KUKA KRL program: paintImage.src, paintImage.dat

--- paintImage.src ---
&ACCESS RVP
&REL 47
DEF paintImage( )
;FOLD Declaration
   DECL EKI_STATUS RET
   DECL FRAME nextPoint
   DECL INT status
   DECL INT currentColor
   DECL BOOL pathStart
   $FLAG[1]=FALSE



   ;FOLD INI;%{PE}
      ;FOLD BASISTECH INI
         GLOBAL INTERRUPT DECL 3 WHEN $STOPMESS==TRUE DO IR_STOPM ( )
         INTERRUPT ON 3
         BAS (#INITMOV,0 )
      ;ENDFOLD (BASISTECH INI)
      ;FOLD USER INI
         ;Make your modifications here

      ;ENDFOLD (USER INI)
      ;ENDFOLD (INI)
      ;FOLD Initialize sample data
         nextPoint = {X 200,Y 600,Z 600}
         status = 0
         currentColor = 1000
         pathStart = TRUE

      ;ENDFOLD (Initialize sample data)
      ;ENDFOLD (Declaration)


   ;FOLD PTP HOME  Vel= 100 % DEFAULT;%{PE}%MKUKATPBASIS,%CMOVE,%VPTP,%P 1:PTP, 2:HOME, 3:, 5:100, 7:DEFAULT
      $BWDSTART = FALSE
      PDAT_ACT=PDEFAULT
      FDAT_ACT=FHOME
      BAS (#PTP_PARAMS,10 )
      $H_POS=XHOME
      PTP  XHOME
   ;ENDFOLD


;FOLD PTP P8 Vel=10 % PDAT4 Tool[2]:pinselC Base[3]:canvas1;%{PE}%R 8.3.48,%MKUKATPBASIS,%CMOVE,%VPTP,%P 1:PTP, 2:P8, 3:, 5:10, 7:PDAT4
$BWDSTART=FALSE
PDAT_ACT=PPDAT4
FDAT_ACT=FP8
BAS(#PTP_PARAMS,10)
PTP XP8
;ENDFOLD
RET=EKI_Init("xmlPaintImage")
RET=EKI_Open("xmlPaintImage")

LOOP
WAIT FOR $FLAG[993] == TRUE
RET=EKI_GetInt("xmlPaintImage","Ext/Status",status)
$FLAG[993] = FALSE

WAIT FOR $FLAG[997] == TRUE

SWITCH status

CASE POINT
RET=EKI_GetFrame("xmlPaintImage","Ext/Points/xyzabc",nextPoint)
if pathStart == TRUE THEN

   ;FOLD PTP hoverNextPoint Vel=20 % PDAT8 Tool[2]:pinselC Base[3]:canvas1;%{PE}%R 8.3.48,%MKUKATPBASIS,%CMOVE,%VPTP,%P 1:PTP, 2:P4, 3:, 5:100, 7:PDAT4
   $BWDSTART=FALSE
   PDAT_ACT=PPDAT2
   FDAT_ACT=FP4
   BAS(#PTP_PARAMS,20)
   PTP nextPoint : {X 0,Y 0,Z -100,A 0,B 0,C 0}
   ;ENDFOLD

   ;FOLD PTP nextPoint Vel=5 % PDAT4 Tool[2]:pinselC Base[3]:canvas1;%{PE}%R 8.3.48,%MKUKATPBASIS,%CMOVE,%VPTP,%P 1:PTP, 2:P4, 3:, 5:100, 7:PDAT4
   $BWDSTART=FALSE
   PDAT_ACT=PPDAT4
   FDAT_ACT=FP4
   BAS(#PTP_PARAMS,5)
   LIN nextPoint
   ;ENDFOLD
   pathStart = FALSE

ENDIF
pathStart = FALSE
;FOLD PTP P4 Vel=100 % PDAT4 Tool[2]:pinselC Base[3]:canvas1;%{PE}%R 8.3.48,%MKUKATPBASIS,%CMOVE,%VPTP,%P 1:PTP, 2:P4, 3:, 5:100, 7:PDAT4
$BWDSTART=FALSE
PDAT_ACT=PPDAT4
FDAT_ACT=FP4
BAS(#PTP_PARAMS,70)
LIN nextPoint
;ENDFOLD


CASE RENEWCOLOR
RET=EKI_GetInt("xmlPaintImage","Ext/Color",currentColor)
pathStart = TRUE
;RET=EKI_GetFrame("xmlPaintImage","Ext/Points/xyzabc",nextPoint)
;FOLD PTP hoverPoint Vel=20 % PDAT4 Tool[2]:pinselC Base[3]:canvas1;%{PE}%R 8.3.48,%MKUKATPBASIS,%CMOVE,%VPTP,%P 1:PTP, 2:P4, 3:, 5:100, 7:PDAT4
$BWDSTART=FALSE
PDAT_ACT=PPDAT4
FDAT_ACT=FP4
BAS(#PTP_PARAMS,20)
PTP $POS_ACT : {X 0,Y 0,Z -100,A 0,B 0,C 0}
;ENDFOLD
colorPick(currentColor)

CASE NEWPATH
RET=EKI_GetFrame("xmlPaintImage","Ext/Points/xyzabc",nextPoint)
pathStart = TRUE
;FOLD PTP hoverPoint Vel=20 % PDAT4 Tool[2]:pinselC Base[3]:canvas1;%{PE}%R 8.3.48,%MKUKATPBASIS,%CMOVE,%VPTP,%P 1:PTP, 2:P4, 3:, 5:100, 7:PDAT4
$BWDSTART=FALSE
PDAT_ACT=PPDAT4
FDAT_ACT=FP4
BAS(#PTP_PARAMS,20)
LIN $POS_ACT : {X 0,Y 0,Z -100,A 0,B 0,C 0}
;ENDFOLD


ENDSWITCH

RET=EKI_ClearBuffer("xmlPaintImage","Ext")
RET=EKI_SetBool("xmlPaintImage","Robot/Status",true)
RET=EKI_Send("xmlPaintImage","Robot")



ENDLOOP

RET=EKI_Clear("xmlPaintImage")
RET=EKI_Close("xmlPaintImage")

   ;FOLD PTP HOME  Vel= 100 % DEFAULT;%{PE}%MKUKATPBASIS,%CMOVE,%VPTP,%P 1:PTP, 2:HOME, 3:, 5:100, 7:DEFAULT
      $BWDSTART = FALSE
      PDAT_ACT=PDEFAULT
      FDAT_ACT=FHOME
      BAS (#PTP_PARAMS,10 )
      $H_POS=XHOME
      PTP  XHOME
   ;ENDFOLD
END

DEF colorPick(COLOR:IN)
INT COLOR
colorHome()
water()
drying()
colorHome()
SWITCH COLOR
   CASE 1
      l1c1()
   CASE 2
      l1c2()
   CASE 3
      l1c3()
   CASE 4
      l2c1()
   CASE 5
      l2c2()
   CASE 6
      l2c3()
   CASE 7
      l3c1()
   CASE 8
      l3c2()
   CASE 9
      l3c3()
   CASE 10
      l4c1()
   CASE 11
      l4c2()
   CASE 12
      l4c3()
ENDSWITCH
colorHome()

END

--- paintImage.dat ---
&ACCESS RVP
&REL 47
DEFDAT  paintImage
;FOLD EXTERNAL DECLARATIONS;%{PE}%MKUKATPBASIS,%CEXT,%VCOMMON,%P
;FOLD BASISTECH EXT;%{PE}%MKUKATPBASIS,%CEXT,%VEXT,%P
EXT  BAS (BAS_COMMAND  :IN,REAL  :IN )
;ENDFOLD (BASISTECH EXT)
;FOLD USER EXT;%{E}%MKUKATPUSER,%CEXT,%VEXT,%P
;Make your modifications here
DECL BOOL collisionocc=FALSE
DECL CONST INT POINT=1
DECL CONST INT RENEWCOLOR=2
DECL CONST INT NEWPATH=3

;ENDFOLD (USER EXT)
;ENDFOLD (EXTERNAL DECLARATIONS)
DECL BASIS_SUGG_T LAST_BASIS={POINT1[] "P10                     ",POINT2[] "P10                     ",CP_PARAMS[] "CPDAT0                  ",PTP_PARAMS[] "PDAT7                   ",CONT[] "                        ",CP_VEL[] "2.0                     ",PTP_VEL[] "20                      ",SYNC_PARAMS[] "SYNCDAT                 ",SPL_NAME[] "S0                      ",A_PARAMS[] "ADAT0                   "}
DECL E6POS XP1={X 272.500458,Y 64.1022873,Z -139.427612,A 88.7173233,B 6.68055201,C -6.75402117,S 2,T 11,E1 0.0,E2 0.0,E3 0.0,E4 0.0,E5 0.0,E6 0.0}
DECL FDAT FP1={TOOL_NO 2,BASE_NO 3,IPO_FRAME #BASE,POINT2[] " ",TQ_STATE FALSE}
DECL PDAT PPDAT2={VEL 100.000,ACC 30.0000,APO_DIST 100.000,GEAR_JERK 10.0000,EXAX_IGN 0}
DECL PDAT PPDAT3={VEL 100.000,ACC 50.0000,APO_DIST 100.000,GEAR_JERK 50.0000,EXAX_IGN 0}
DECL E6POS XP2={X 272.500458,Y 64.1022873,Z -139.427612,A 88.7173233,B 6.68055201,C -6.75402117,S 2,T 11,E1 0.0,E2 0.0,E3 0.0,E4 0.0,E5 0.0,E6 0.0}
DECL FDAT FP2={TOOL_NO 2,BASE_NO 3,IPO_FRAME #BASE,POINT2[] " ",TQ_STATE FALSE}
DECL E6POS XP3={X 323.515778,Y 71.6573486,Z -150.640778,A 88.7295532,B 6.69334459,C -15.0158014,S 2,T 10,E1 0.0,E2 0.0,E3 0.0,E4 0.0,E5 0.0,E6 0.0}
DECL FDAT FP3={TOOL_NO 2,BASE_NO 3,IPO_FRAME #BASE,POINT2[] " ",TQ_STATE FALSE}
DECL PDAT PPDAT4={VEL 100.000,ACC 50.0000,APO_DIST 100.000,GEAR_JERK 50.0000,EXAX_IGN 0}
DECL E6POS XP4={X 323.515778,Y 71.6573486,Z -150.640778,A 88.7295532,B 6.69334459,C -15.0158014,S 2,T 10,E1 0.0,E2 0.0,E3 0.0,E4 0.0,E5 0.0,E6 0.0}
DECL FDAT FP4={TOOL_NO 2,BASE_NO 3,IPO_FRAME #BASE,POINT2[] " ",TQ_STATE FALSE}
DECL E6POS XP5={X 1347.12073,Y 37.7801933,Z 1062.70044,A -107.690994,B 42.5165787,C -105.567268,S 2,T 3,E1 0.0,E2 0.0,E3 0.0,E4 0.0,E5 0.0,E6 0.0}
DECL FDAT FP5={TOOL_NO 2,BASE_NO 5,IPO_FRAME #BASE,POINT2[] " ",TQ_STATE FALSE}
DECL PDAT PPDAT5={VEL 100.000,ACC 100.000,APO_DIST 100.000,GEAR_JERK 50.0000,EXAX_IGN 0}
DECL E6POS XP6={X 1347.12073,Y 37.7801933,Z 1062.70044,A -107.690994,B 42.5165787,C -105.567268,S 2,T 3,E1 0.0,E2 0.0,E3 0.0,E4 0.0,E5 0.0,E6 0.0}
DECL FDAT FP6={TOOL_NO 2,BASE_NO 5,IPO_FRAME #BASE,POINT2[] " ",TQ_STATE FALSE}
DECL E6POS XP7={X 1347.12073,Y 37.7801933,Z 1062.70044,A -107.690994,B 42.5165787,C -105.567268,S 2,T 3,E1 0.0,E2 0.0,E3 0.0,E4 0.0,E5 0.0,E6 0.0}
DECL FDAT FP7={TOOL_NO 2,BASE_NO 5,IPO_FRAME #BASE,POINT2[] " ",TQ_STATE FALSE}
DECL E6POS XP8={X 109.677643,Y -6.88640451,Z -63.7406158,A 46.4953041,B 9.04451,C -5.17782068,S 2,T 3,E1 0.0,E2 0.0,E3 0.0,E4 0.0,E5 0.0,E6 0.0}
DECL FDAT FP8={TOOL_NO 2,BASE_NO 3,IPO_FRAME #BASE,POINT2[] " ",TQ_STATE FALSE}
DECL PDAT PPDAT6={VEL 100.000,ACC 50.0000,APO_DIST 100.000,GEAR_JERK 50.0000,EXAX_IGN 0}
DECL E6POS XP9={X 323.515778,Y 71.6573486,Z -150.640778,A 88.7295532,B 6.69334459,C -15.0158014,S 2,T 10,E1 0.0,E2 0.0,E3 0.0,E4 0.0,E5 0.0,E6 0.0}
DECL FDAT FP9={TOOL_NO 2,BASE_NO 3,IPO_FRAME #BASE,POINT2[] " ",TQ_STATE FALSE}
DECL PDAT PPDAT7={VEL 100.000,ACC 50.0000,APO_DIST 100.000,GEAR_JERK 50.0000,EXAX_IGN 0}
DECL E6POS XP10={X 323.515778,Y 71.6573486,Z -150.640778,A 88.7295532,B 6.69334459,C -15.0158014,S 2,T 10,E1 0.0,E2 0.0,E3 0.0,E4 0.0,E5 0.0,E6 0.0}
DECL FDAT FP10={TOOL_NO 2,BASE_NO 3,IPO_FRAME #BASE,POINT2[] " ",TQ_STATE FALSE}
ENDDAT
